Yaskawa INFORM job: R1_W53-A1(90,180)R2.JBI

/JOB
//NAME R1_W53-A1(90,180)R2
///FOLDERNAME KRIS-SCIANA
//POS
///NPOS 55,55,0,2,0,0
///TOOL 0
///POSTYPE PULSE
///PULSE
C00000=-4393,39408,-45850,-56974,107866,-38635
C00001=-4393,39408,-45850,-56974,107866,-38635
C00002=-57127,104326,11609,-56974,107866,-38635
C00003=-57127,77996,9631,-53904,100642,-33810
C00004=-68868,97406,33308,-40326,102880,-35891
C00005=-82230,129861,77644,-13538,109090,-35165
C00006=-74204,109555,58440,-31590,104867,-34569
C00007=-74418,111138,60545,-31493,104377,-34509
C00008=-74011,108607,56192,-31755,105702,-34736
C00009=-74506,112378,60945,-31547,104681,-34629
C00010=-74506,112095,61194,-31498,104425,-34555
C00011=-74506,112776,60621,-31611,105028,-34729
C00012=-77451,100941,50515,-32929,89610,-16321
C00013=-77412,99737,49701,-32937,89525,-16280
C00014=-80659,92020,40491,-24215,87124,-15265
C00015=-80482,93141,41920,-24275,86894,-15157
C00016=-77163,100530,53168,-32990,88157,-15788
C00017=-76618,101794,49218,-33172,90958,-16406
C00018=-76874,111247,51005,-11099,107559,11799
C00019=-80591,101914,38375,-2703,106264,12355
C00020=-80592,99641,39044,-2679,104686,12390
C00021=-78963,101321,42944,-5743,104646,12327
C00022=-80323,96551,37168,-2714,104262,12484
C00023=-80415,98263,37603,-2708,104870,12441
C00024=-74390,114145,60912,1929,95252,15443
C00025=-76720,104512,45399,2277,100139,14322
C00026=-80580,101336,38397,2674,103460,12021
C00027=-78782,133634,80935,-13996,103384,75839
C00028=-74724,95428,37925,-23998,105933,75088
C00029=-74934,121529,74207,-18787,109795,75838
C00030=-71821,116038,70063,-18565,110218,76919
C00031=-72430,124724,76841,-18643,110363,76670
C00032=-74362,69960,2524,-6218,105815,36629
C00033=-69157,63041,7727,-10776,93973,38093
C00034=-69752,61654,6114,-10607,94178,37894
C00035=-73709,53321,-3394,-9465,95292,36609
C00036=-75219,53872,-3292,-7232,98435,36398
C00037=-74402,58837,-4462,-7542,101743,36441
C00038=-77887,57064,-12764,-6743,105659,35208
C00039=-73093,75194,9445,-23568,108624,22498
C00040=-73093,75194,9445,-23568,108624,47779
C00041=-74905,65081,7445,-31390,103058,39674
C00042=-72301,70815,16458,-32002,102536,41501
C00043=-69710,70391,12700,-33158,105675,42200
C00044=-73972,83218,17017,-18195,115594,43024
C00045=-73978,83090,16854,-18172,115571,194
C00046=-76924,77433,14323,-17678,113737,-498
C00047=-73877,53266,-6769,-20778,100180,1705
C00048=-76780,55069,-4744,-19948,99266,960
C00049=-75630,59436,179,-22898,101050,4210
C00050=-73226,63195,7664,-34213,103404,1761
C00051=-68667,65027,2719,-35925,108314,1828
C00052=-76429,130747,61875,-15141,113703,75346
C00053=-76429,130747,61875,-14899,59891,75343
C00054=-26986,34352,-63131,-44278,95581,80088
BC00000=14738,708513,1064454
BC00001=14738,708513,1064454
BC00002=14738,708513,1064454
BC00003=14738,708513,1064454
BC00004=14738,708513,1064454
BC00005=14737,708513,1064458
BC00006=14737,708513,1064458
BC00007=14737,708513,1064458
BC00008=14737,708513,1064458
BC00009=14737,708513,1064458
BC00010=14737,708513,1064458
BC00011=14737,708513,1064458
BC00012=21248,678730,1064458
BC00013=21262,675288,1064458
BC00014=21262,675288,1064458
BC00015=21262,675288,1064458
BC00016=21262,675288,1064458
BC00017=21262,675288,1064458
BC00018=139,705625,1064458
BC00019=139,705625,1064458
BC00020=628,709764,1064458
BC00021=679,710198,1064458
BC00022=823,711419,1064458
BC00023=823,711419,1064458
BC00024=679,710198,1064458
BC00025=8500,710301,1064458
BC00026=26280,706465,1064458
BC00027=25958,706513,1064458
BC00028=25958,722166,1064458
BC00029=25958,722166,1064458
BC00030=25958,722166,1064458
BC00031=25958,722166,1064458
BC00032=25958,722166,1064458
BC00033=27551,915714,1084352
BC00034=27551,915714,1084352
BC00035=27551,915714,1084352
BC00036=27551,915714,1084352
BC00037=27551,915714,1084352
BC00038=25958,722166,1064458
BC00039=25958,722166,1064458
BC00040=25958,722166,1064458
BC00041=25958,722166,1064458
BC00042=25959,722166,1064456
BC00043=25958,722165,1064456
BC00044=25958,722165,1064456
BC00045=25958,722165,1064456
BC00046=25958,722165,1064456
BC00047=25958,722165,1064456
BC00048=25958,722165,1064456
BC00049=25958,722165,1064456
BC00050=25958,722165,1064456
BC00051=25958,722165,1064456
BC00052=25958,706513,1064458
BC00053=25958,665434,1064458
BC00054=25958,667245,1064458
///POSTYPE BASE
///RECTAN
///RCONF 0,0,0,0,0,0,0,0,0,0,0,0,0,0,0,0,0,0,0,0,0,0,0,0
P00006=0.222,-3.123,-1.508,0.0000,0.0000,0.0000
P00022=0.222,-3.123,-1.508,0.0000,0.0000,0.0000
//INST
///DATE 2024/07/25 11:33
///ATTR SC,RW
///GROUP1 RB1,BS1
NOP
'r2_W53-A1(90,180)
'Path S1056
SFTOF
MOVJ C00000 BC00000 VJ=50.00
MOVJ C00001 BC00001 VJ=20.00
MOVJ C00002 BC00002 VJ=10.00
MOVJ C00003 BC00003 VJ=20.00
MOVJ C00004 BC00004 VJ=20.00
MOVL C00005 BC00005 V=100.0
MOVL C00006 BC00006 V=60.0
REFP 3 C00007 BC00007
CALL JOB:SEARCH-R1
SET P022 P006
SFTON P022
MOVL C00008 BC00008 V=166.7
MOVL C00009 BC00009 V=166.7
REFP 3 C00010 BC00010
CALL JOB:SEARCH-R1
SET P022 P006
SFTON P022
MOVL C00011 BC00011 V=100.0
MOVL C00012 BC00012 V=100.0
MOVL C00013 BC00013 V=60.0
MOVL C00014 BC00014 V=60.0
REFP 3 C00015 BC00015
CALL JOB:SEARCH-R1
SET P022 P006
SFTON P022
MOVL C00016 BC00016 V=60.0
MOVL C00017 BC00017 V=100.0
'Path W1057
SFTOF
SFTON P022
MOVJ C00018 BC00018 VJ=20.00
MOVJ C00019 BC00019 VJ=20.00 PL=0
MOVL C00020 BC00020 V=100.0
MOVL C00021 BC00021 V=100.0 PL=0
REFP 1 C00022 BC00022
REFP 2 C00023 BC00023
MACRO1 MJ#(0) ARGF6
ARCON
MOVL C00024 BC00024 V=10.0
ARCOF
MOVL C00025 BC00025 V=166.7
MOVL C00026 BC00026 V=166.7
SFTOF
SFTON P022
'COMMENT
MOVJ C00027 BC00027 VJ=20.00
MOVL C00028 BC00028 V=100.0 PL=0
MACRO1 MJ#(0) ARGF6
ARCON
MOVL C00029 BC00029 V=8.3
MOVL C00030 BC00030 V=8.3
ARCOF
MOVL C00031 BC00031 V=166.7
MOVL C00032 BC00032 V=166.7
COMM MACRO1 MJ#(0) ARGF6
COMM MOVL C00033 BC00033 V=83.3
COMM ARCON
COMM MOVL C00034 BC00034 V=10.0
COMM MOVL C00035 BC00035 V=10.0
COMM MOVL C00036 BC00036 V=10.0
COMM ARCOF
COMM MOVJ C00037 BC00037 VJ=10.00
MOVJ C00038 BC00038 VJ=10.00
MOVJ C00039 BC00039 VJ=10.00
MOVJ C00040 BC00040 VJ=10.00
MACRO1 MJ#(0) ARGF7
MOVJ C00041 BC00041 VJ=10.00
ARCON
MOVL C00042 BC00042 V=8.3
ARCOF
MOVJ C00043 BC00043 VJ=10.00
MOVJ C00044 BC00044 VJ=10.00
MOVJ C00045 BC00045 VJ=10.00
MOVJ C00046 BC00046 VJ=10.00
MOVJ C00047 BC00047 VJ=10.00
ARCON
MOVL C00048 BC00048 V=10.0
MOVL C00049 BC00049 V=10.0
MOVL C00050 BC00050 V=10.0
ARCOF
MOVJ C00051 BC00051 VJ=10.00
MOVJ C00052 BC00052 VJ=40.00
MOVJ C00053 BC00053 VJ=100.00
SFTOF
MOVJ C00054 BC00054 VJ=100.00
END
